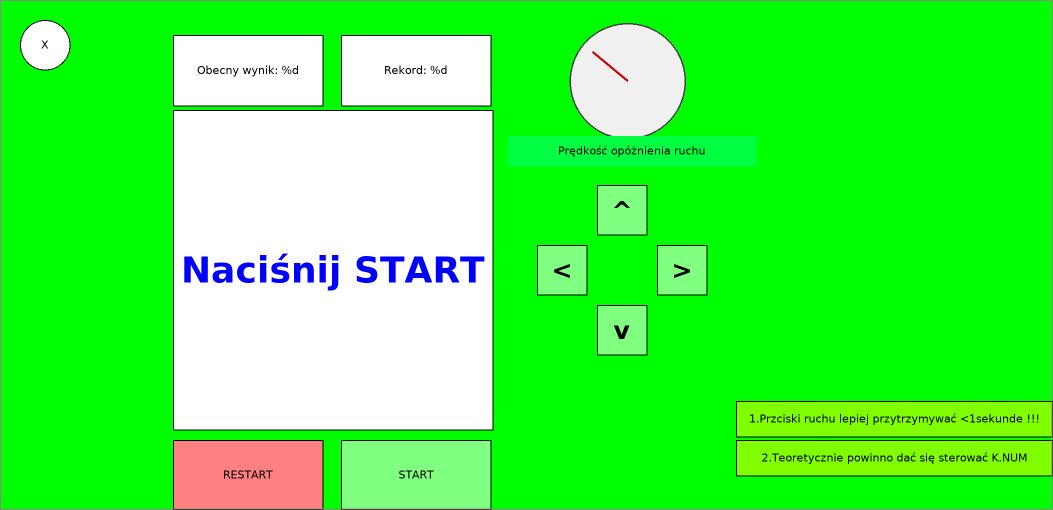
VISUALIZATION Snake  // 1053x510
    Rectangle (173,110 30x30), colour toggle: MAIN.gra.poleGry.MacierzPola[1][1]
    Rectangle (205,110 30x30), colour toggle: MAIN.gra.poleGry.MacierzPola[1][2]
    Rectangle (173,142 30x30), colour toggle: MAIN.gra.poleGry.MacierzPola[2][1]
    Rectangle (173,174 30x30), colour toggle: MAIN.gra.poleGry.MacierzPola[3][1]
    Rectangle (173,206 30x30), colour toggle: MAIN.gra.poleGry.MacierzPola[4][1]
    Rectangle (173,238 30x30), colour toggle: MAIN.gra.poleGry.MacierzPola[5][1]
    Rectangle (173,270 30x30), colour toggle: MAIN.gra.poleGry.MacierzPola[6][1]
    Rectangle (173,302 30x30), colour toggle: MAIN.gra.poleGry.MacierzPola[7][1]
    Rectangle (173,334 30x30), colour toggle: MAIN.gra.poleGry.MacierzPola[8][1]
    Rectangle (173,366 30x30), colour toggle: MAIN.gra.poleGry.MacierzPola[9][1]
    Rectangle (173,398 30x30), colour toggle: MAIN.gra.poleGry.MacierzPola[10][1]
    Rectangle (237,110 30x30), colour toggle: MAIN.gra.poleGry.MacierzPola[1][3]
    Rectangle (269,110 30x30), colour toggle: MAIN.gra.poleGry.MacierzPola[1][4]
    Rectangle (301,110 30x30), colour toggle: MAIN.gra.poleGry.MacierzPola[1][5]
    Rectangle (333,110 30x30), colour toggle: MAIN.gra.poleGry.MacierzPola[1][6]
    Rectangle (365,110 30x30), colour toggle: MAIN.gra.poleGry.MacierzPola[1][7]
    Rectangle (397,110 30x30), colour toggle: MAIN.gra.poleGry.MacierzPola[1][8]
    Rectangle (429,110 30x30), colour toggle: MAIN.gra.poleGry.MacierzPola[1][9]
    Rectangle (461,110 30x30), colour toggle: MAIN.gra.poleGry.MacierzPola[1][10]
    Rectangle (205,142 30x30), colour toggle: MAIN.gra.poleGry.MacierzPola[2][2]
    Rectangle (237,142 30x30), colour toggle: MAIN.gra.poleGry.MacierzPola[2][3]
    Rectangle (269,142 30x30), colour toggle: MAIN.gra.poleGry.MacierzPola[2][4]
    Rectangle (301,142 30x30), colour toggle: MAIN.gra.poleGry.MacierzPola[2][5]
    Rectangle (333,142 30x30), colour toggle: MAIN.gra.poleGry.MacierzPola[2][6]
    Rectangle (365,142 30x30), colour toggle: MAIN.gra.poleGry.MacierzPola[2][7]
    Rectangle (397,142 30x30), colour toggle: MAIN.gra.poleGry.MacierzPola[2][8]
    Rectangle (429,142 30x30), colour toggle: MAIN.gra.poleGry.MacierzPola[2][9]
    Rectangle (461,142 30x30), colour toggle: MAIN.gra.poleGry.MacierzPola[2][10]
    Rectangle (205,174 30x30), colour toggle: MAIN.gra.poleGry.MacierzPola[3][2]
    Rectangle (237,174 30x30), colour toggle: MAIN.gra.poleGry.MacierzPola[3][3]
    Rectangle (269,174 30x30), colour toggle: MAIN.gra.poleGry.MacierzPola[3][4]
    Rectangle (301,174 30x30), colour toggle: MAIN.gra.poleGry.MacierzPola[3][5]
    Rectangle (333,174 30x30), colour toggle: MAIN.gra.poleGry.MacierzPola[3][6]
    Rectangle (365,174 30x30), colour toggle: MAIN.gra.poleGry.MacierzPola[3][7]
    Rectangle (397,174 30x30), colour toggle: MAIN.gra.poleGry.MacierzPola[3][8]
    Rectangle (429,174 30x30), colour toggle: MAIN.gra.poleGry.MacierzPola[3][9]
    Rectangle (461,174 30x30), colour toggle: MAIN.gra.poleGry.MacierzPola[3][10]
    Rectangle (205,206 30x30), colour toggle: MAIN.gra.poleGry.MacierzPola[4][2]
    Rectangle (237,206 30x30), colour toggle: MAIN.gra.poleGry.MacierzPola[4][3]
    Rectangle (269,206 30x30), colour toggle: MAIN.gra.poleGry.MacierzPola[4][4]
    Rectangle (301,206 30x30), colour toggle: MAIN.gra.poleGry.MacierzPola[4][5]
    Rectangle (333,206 30x30), colour toggle: MAIN.gra.poleGry.MacierzPola[4][6]
    Rectangle (365,206 30x30), colour toggle: MAIN.gra.poleGry.MacierzPola[4][7]
    Rectangle (397,206 30x30), colour toggle: MAIN.gra.poleGry.MacierzPola[4][8]
    Rectangle (429,206 30x30), colour toggle: MAIN.gra.poleGry.MacierzPola[4][9]
    Rectangle (461,206 30x30), colour toggle: MAIN.gra.poleGry.MacierzPola[4][10]
    Rectangle (205,238 30x30), colour toggle: MAIN.gra.poleGry.MacierzPola[5][2]
    Rectangle (237,238 30x30), colour toggle: MAIN.gra.poleGry.MacierzPola[5][3]
    Rectangle (269,238 30x30), colour toggle: MAIN.gra.poleGry.MacierzPola[5][4]
    Rectangle (301,238 30x30), colour toggle: MAIN.gra.poleGry.MacierzPola[5][5]
    Rectangle (333,238 30x30), colour toggle: MAIN.gra.poleGry.MacierzPola[5][6]
    Rectangle (365,238 30x30), colour toggle: MAIN.gra.poleGry.MacierzPola[5][7]
    Rectangle (397,238 30x30), colour toggle: MAIN.gra.poleGry.MacierzPola[5][8]
    Rectangle (429,238 30x30), colour toggle: MAIN.gra.poleGry.MacierzPola[5][9]
    Rectangle (461,238 30x30), colour toggle: MAIN.gra.poleGry.MacierzPola[5][10]
    Rectangle (205,270 30x30), colour toggle: MAIN.gra.poleGry.MacierzPola[6][2]
    Rectangle (237,270 30x30), colour toggle: MAIN.gra.poleGry.MacierzPola[6][3]
    Rectangle (269,270 30x30), colour toggle: MAIN.gra.poleGry.MacierzPola[6][4]
    Rectangle (301,270 30x30), colour toggle: MAIN.gra.poleGry.MacierzPola[6][5]
    Rectangle (333,270 30x30), colour toggle: MAIN.gra.poleGry.MacierzPola[6][6]
    Rectangle (365,270 30x30), colour toggle: MAIN.gra.poleGry.MacierzPola[6][7]
    Rectangle (397,270 30x30), colour toggle: MAIN.gra.poleGry.MacierzPola[6][8]
    Rectangle (429,270 30x30), colour toggle: MAIN.gra.poleGry.MacierzPola[6][9]
    Rectangle (461,270 30x30), colour toggle: MAIN.gra.poleGry.MacierzPola[6][10]
    Rectangle (205,302 30x30), colour toggle: MAIN.gra.poleGry.MacierzPola[7][2]
    Rectangle (237,302 30x30), colour toggle: MAIN.gra.poleGry.MacierzPola[7][3]
    Rectangle (269,302 30x30), colour toggle: MAIN.gra.poleGry.MacierzPola[7][4]
    Rectangle (301,302 30x30), colour toggle: MAIN.gra.poleGry.MacierzPola[7][5]
    Rectangle (333,302 30x30), colour toggle: MAIN.gra.poleGry.MacierzPola[7][6]
    Rectangle (365,302 30x30), colour toggle: MAIN.gra.poleGry.MacierzPola[7][7]
    Rectangle (397,302 30x30), colour toggle: MAIN.gra.poleGry.MacierzPola[7][8]
    Rectangle (429,302 30x30), colour toggle: MAIN.gra.poleGry.MacierzPola[7][9]
    Rectangle (461,302 30x30), colour toggle: MAIN.gra.poleGry.MacierzPola[7][10]
    Rectangle (205,334 30x30), colour toggle: MAIN.gra.poleGry.MacierzPola[8][2]
    Rectangle (237,334 30x30), colour toggle: MAIN.gra.poleGry.MacierzPola[8][3]
    Rectangle (269,334 30x30), colour toggle: MAIN.gra.poleGry.MacierzPola[8][4]
    Rectangle (301,334 30x30), colour toggle: MAIN.gra.poleGry.MacierzPola[8][5]
    Rectangle (333,334 30x30), colour toggle: MAIN.gra.poleGry.MacierzPola[8][6]
    Rectangle (365,334 30x30), colour toggle: MAIN.gra.poleGry.MacierzPola[8][7]
    Rectangle (397,334 30x30), colour toggle: MAIN.gra.poleGry.MacierzPola[8][8]
    Rectangle (429,334 30x30), colour toggle: MAIN.gra.poleGry.MacierzPola[8][9]
    Rectangle (461,334 30x30), colour toggle: MAIN.gra.poleGry.MacierzPola[8][10]
    Rectangle (205,366 30x30), colour toggle: MAIN.gra.poleGry.MacierzPola[9][2]
    Rectangle (237,366 30x30), colour toggle: MAIN.gra.poleGry.MacierzPola[9][3]
    Rectangle (269,366 30x30), colour toggle: MAIN.gra.poleGry.MacierzPola[9][4]
    Rectangle (301,366 30x30), colour toggle: MAIN.gra.poleGry.MacierzPola[9][5]
    Rectangle (333,366 30x30), colour toggle: MAIN.gra.poleGry.MacierzPola[9][6]
    Rectangle (365,366 30x30), colour toggle: MAIN.gra.poleGry.MacierzPola[9][7]
    Rectangle (397,366 30x30), colour toggle: MAIN.gra.poleGry.MacierzPola[9][8]
    Rectangle (429,366 30x30), colour toggle: MAIN.gra.poleGry.MacierzPola[9][9]
    Rectangle (461,366 30x30), colour toggle: MAIN.gra.poleGry.MacierzPola[9][10]
    Rectangle (205,398 30x30), colour toggle: MAIN.gra.poleGry.MacierzPola[10][2]
    Rectangle (237,398 30x30), colour toggle: MAIN.gra.poleGry.MacierzPola[10][3]
    Rectangle (269,398 30x30), colour toggle: MAIN.gra.poleGry.MacierzPola[10][4]
    Rectangle (301,398 30x30), colour toggle: MAIN.gra.poleGry.MacierzPola[10][5]
    Rectangle (333,398 30x30), colour toggle: MAIN.gra.poleGry.MacierzPola[10][6]
    Rectangle (365,398 30x30), colour toggle: MAIN.gra.poleGry.MacierzPola[10][7]
    Rectangle (397,398 30x30), colour toggle: MAIN.gra.poleGry.MacierzPola[10][8]
    Rectangle (429,398 30x30), colour toggle: MAIN.gra.poleGry.MacierzPola[10][9]
    Rectangle (461,398 30x30), colour toggle: MAIN.gra.poleGry.MacierzPola[10][10]
    Ellipse (20,20 50x50), "X"
        OnMouseClick: change screen: EkranGlowny
    RoundedRectangle (173,440 150x70), "RESTART", colour toggle: GVL_Lista.bStanPrzyciskuRestart
        OnMouseDown: toggle GVL_Lista.bStanPrzyciskuRestart
        OnMouseUp: toggle GVL_Lista.bStanPrzyciskuRestart
    Rectangle (537,245 50x50), "<"
        OnMouseDown: toggle GVL_Lista.bStanStrzalek[1]
        OnMouseUp: toggle GVL_Lista.bStanStrzalek[1]
    Rectangle (597,305 50x50), "v"
        OnMouseDown: toggle GVL_Lista.bStanStrzalek[2]
        OnMouseUp: toggle GVL_Lista.bStanStrzalek[2]
    Rectangle (657,245 50x50), ">"
        OnMouseDown: toggle GVL_Lista.bStanStrzalek[3]
        OnMouseUp: toggle GVL_Lista.bStanStrzalek[3]
    Rectangle (597,185 50x50), "^"
        OnMouseDown: toggle GVL_Lista.bStanStrzalek[4]
        OnMouseUp: toggle GVL_Lista.bStanStrzalek[4]
    RoundedRectangle (173,35 150x71), "Obecny wynik: %d", text variable: MAIN.gra.iLicnikPunktow
    RoundedRectangle (341,35 150x71), "Rekord: %d", text variable: GVL_Lista.iRekord
    Rectangle (173,110 320x320), "KONIEC GRY", invisible if: MAIN.gra.GAMEOVER
    Rectangle (173,110 320x320), "Naciśnij START", invisible if: MAIN.gra.EKRANSTARTOWY
    RoundedRectangle (341,440 150x70), "START", colour toggle: GVL_Lista.bStanPRzyciskuStartu
        OnMouseDown: toggle GVL_Lista.bStanPRzyciskuStartu
        OnMouseUp: toggle GVL_Lista.bStanPRzyciskuStartu
    Meter180 (516,23 223x116), value: MAIN.gra.timerRuchu.PT, style: Meter-Meter180-Gray, scale format: %.1f, scale 0..1000
        p518627256: ms
    Rectangle (508,136 248x30), "Prędkość opóżnienia ruchu"
    Rectangle (736,401 317x36), "1.Przciski ruchu lepiej przytrzymywać <1sekunde !!!"
    Rectangle (736,440 317x36), "2.Teoretycznie powinno dać się sterować K.NUM"
    hotkey HotkeyInput Id=481047871488, Key=KeyDown=True, KeyName=8, VisuElemId=275
    hotkey HotkeyInput Id=481048920064, Key=KeyName=8, VisuElemId=275
    hotkey HotkeyInput Id=481049968640, Key=KeyDown=True, KeyName=4, VisuElemId=263
    hotkey HotkeyInput Id=481051017216, Key=KeyName=4, VisuElemId=263
    hotkey HotkeyInput Id=481052065792, Key=KeyDown=True, KeyName=6, VisuElemId=273
    hotkey HotkeyInput Id=481053114368, Key=KeyName=6, VisuElemId=273
    hotkey HotkeyInput Id=481054162944, Key=KeyDown=True, KeyName=2, VisuElemId=271
    hotkey HotkeyInput Id=481055211520, Key=KeyName=2, VisuElemId=271
END_VISUALIZATION

(* stored: Version 1.1.0.1, ProductVersion 3.1.4024.4
   Visu Snake: Id {e731cc30-2b46-4686-a185-cf9f58a88804} *)
